{attribute 'qualified_only'}
{attribute 'strict'}
TYPE BagCmd:
(
	DO_NOTHING := 0,
    INSERT_BAG_HOLDER := 1,
    REMOVE_BAG_HOLDER := 2
);
END_TYPE

(* stored: Version 1.1.0.1, ProductVersion 3.1.4024.12
   DUT BagCmd: Id {4faa6746-5de0-4cb6-a6c4-3656231adfa9} *)
